FUNCTION_BLOCK TagCmp IMPLEMENTS I_TagCmp
VAR
	_iBaseTag		: I_Tag;
	_eResult		: Results.Result;
	_bLock			: BOOL;
END_VAR

PROPERTY PRIVATE _self : I_TagCmp
GET
VAR
	_this : I_TagCmp := THIS^;
END_VAR
_self := _this;
END_GET
END_PROPERTY

METHOD AndIf : I_TagCmp
VAR_INPUT
	bCondition: BOOL;
END_VAR
AndIf := _self;

IF _bLock THEN
	RETURN;
END_IF

IF _eResult = Results.Ok AND_THEN bCondition THEN
	_eResult := Results.Ok;
END_IF
END_METHOD

METHOD Default : BOOL
IF _bLock THEN
	RETURN;
END_IF

IF _eResult <> Results.None THEN
	RETURN;
END_IF

_bLock := TRUE;
Default := TRUE;
END_METHOD

METHOD IsErr : BOOL
IF _bLock THEN
	RETURN;
END_IF

IF _eResult >= 0 THEN
	RETURN;
END_IF

_bLock := TRUE;
IsErr := TRUE;
END_METHOD

METHOD IsOk : BOOL
IF _bLock THEN
	RETURN;
END_IF

IF _eResult <> Results.Ok THEN
	RETURN;
END_IF

_bLock := TRUE;
IsOk := TRUE;
END_METHOD

METHOD Match : I_TagCmp
VAR_INPUT
	iOther: I_Tag;
END_VAR
Match := _self;

IF _bLock THEN
	RETURN;
END_IF

CASE _eResult OF
	Results.Ok,
	Results.None:
		IF iOther = _iBaseTag THEN
			_eResult := Results.Ok;
		END_IF
END_CASE
END_METHOD

METHOD MatchId : I_TagCmp
VAR_INPUT
	sOtherId	: Strings.Str;
END_VAR
MatchId := _self;

IF _bLock THEN
	RETURN;
END_IF

CASE _eResult OF
	Results.Ok,
	Results.None:
		IF sOtherId <> '' AND_THEN _iBaseTag.GetId() = sOtherId THEN
			_eResult := Results.Ok;
		END_IF
END_CASE
END_METHOD

METHOD MatchPrtId : I_TagCmp
VAR_INPUT
	sPartialId		: Strings.Str;
END_VAR
MatchPrtId := _self;

IF _bLock THEN
	RETURN;
END_IF

CASE _eResult OF
	Results.Ok,
	Results.None:
		IF sPartialId <> '' AND_THEN (Tc2_Standard.RIGHT(_iBaseTag.GetId(), Tc2_Standard.LEN(sPartialId)) = sPartialId) THEN
			_eResult := Results.Ok;
		END_IF
END_CASE
END_METHOD

METHOD OrIf : I_TagCmp
VAR_INPUT
	bCondition: BOOL;
END_VAR
OrIf := _self;

IF _bLock THEN
	RETURN;
END_IF

IF _eResult = Results.Ok OR_ELSE bCondition THEN
	_eResult := Results.Ok;
END_IF
END_METHOD

METHOD Set : I_TagCmp
VAR_INPUT
	iBaseTag	: I_Tag;
END_VAR
_iBaseTag := iBaseTag;
_eResult := Results.None;
_bLock := FALSE;

IF iBaseTag = 0 THEN
	_eResult := Results.Err.Itf0;
END_IF

Set := _self;
END_METHOD

METHOD XorIf : I_TagCmp
VAR_INPUT
	bCondition: BOOL;
END_VAR
XorIf := _self;

IF _bLock THEN
	RETURN;
END_IF

IF _eResult = Results.Ok XOR bCondition THEN
	_eResult := Results.Ok;
END_IF
END_METHOD

END_FUNCTION_BLOCK

(* stored: Version 1.1.0.1
   POU TagCmp: Id {fc472a51-95c8-4c63-b8c5-5dfa13d61d73}, SpecialFunc None
   Property _self: Id {fe4340bb-7f6f-44d0-993a-3f0ac0014f79}
   Get Get: Id {e6bce7a1-dcf6-45e3-9283-e9e637ba0ada}
   Method AndIf: Id {9223b46b-6be4-477a-9010-c0212fbeba73}
   Method Default: Id {4388843a-3f13-4d13-9444-a6c347a1b77c}
   Method IsErr: Id {238cf0db-bccc-4190-9a10-55e053cafa94}
   Method IsOk: Id {1b9b036d-e9fe-45a3-8945-f3ba7babe854}
   Method Match: Id {5c938a28-c260-4bf1-adcc-c84d59421fa8}
   Method MatchId: Id {4a9b5161-c30a-43ce-a366-efe275b3f2b8}
   Method MatchPrtId: Id {78d82c00-f656-4a95-b467-0eabd905f45b}
   Method OrIf: Id {c9bdb97c-3eb5-4133-8ad4-a1531337cf33}
   Method Set: Id {2167daab-4164-44b9-93b7-a85c88a05ebd}
   Method XorIf: Id {ca9c46ad-c94a-433e-aeab-483b4c5ea474} *)
